// TwinCAT 3 PLC project setpositionGen
// ProgramVersion: 3.1.4020.4
// libraries:
//   Tc2_MC2, * (Beckhoff Automation GmbH)
//   Tc2_Standard, * (Beckhoff Automation GmbH)
//   Tc2_System, * (Beckhoff Automation GmbH)
//   Tc2_TcpIp, * (Beckhoff Automation GmbH)
//   Tc3_Module, * (Beckhoff Automation GmbH)
// project tree:
//   DUTs/ state.TcDUT
//   GVLs/ GVL.TcGVL
//   / PlcTask.TcTTO
//   POUs/ MAIN.TcPOU, TCPServer.TcPOU
// real-time tasks:
//   TASK PlcTask: cycle T#4ms, priority 20, ADS port 350
// motion (NC):
//   TASK NC-Task 1 SAF: cycle T#4ms, priority 4, ADS port 501
//   TASK NC-Task 1 SVB: cycle T#2ms, priority 8, ADS port 511
//   AXIS Axis 1 (id 1)
//     General: UnitName=°
//     Dynamic: AccelerationMaximum=75000, DecelerationMaximum=75000, Acceleration=10000, Deceleration=10000, Jerk=2000000
//     Velo: RefSearch=100, RefSync=100, SlowManual=50, Fast=500, Maximum=744
//     PositionAreaControl: Enable=false, Range=360
//     TargetPosControl: Range=360, Time=0.01
//     encoder EncType=19
//       EncPara: ScaleFactorNumerator=360, ScaleFactorDenominator=421888, Inverse=true, MaxCount=#xffffffff
//     drive DrvType=16
//       DrvPara: MaxCount=#xffffffff, DriveControlDWord=#x00020000
//         Analog: VeloReferenz=100, TorqueSetpointScale=10
//         TimeComp: TaskDelayCycles=1
//     controller CtrType=1
//       CtrPara: PriorControlFactor=1
//         PosDiffControl: Enable=false, Range=360
//         Observer: BandWidth=20
//   AXIS Axis 2 (id 2)
//     General: UnitName=°
//     Dynamic: AccelerationMaximum=75000, DecelerationMaximum=75000, Acceleration=10000, Deceleration=10000, Jerk=2000000
//     Velo: RefSearch=100, RefSync=100, SlowManual=50, Fast=500, Maximum=744
//     PositionAreaControl: Enable=false, Range=360
//     TargetPosControl: Range=360, Time=0.01
//     encoder EncType=19
//       EncPara: ScaleFactorNumerator=360, ScaleFactorDenominator=421888, Inverse=true, MaxCount=#xffffffff
//     drive DrvType=16
//       DrvPara: MaxCount=#xffffffff, DriveControlDWord=#x00020000
//         Analog: VeloReferenz=100, TorqueSetpointScale=10
//         TimeComp: TaskDelayCycles=1
//     controller CtrType=1
//       CtrPara: PriorControlFactor=1
//         PosDiffControl: Enable=false, Range=360
//         Observer: BandWidth=20
//   AXIS Axis 3 (id 3)
//     General: UnitName=°
//     Dynamic: AccelerationMaximum=75000, DecelerationMaximum=75000, Acceleration=10000, Deceleration=10000, Jerk=2000000
//     Velo: RefSearch=100, RefSync=100, SlowManual=50, Fast=500, Maximum=744
//     PositionAreaControl: Enable=false, Range=360
//     TargetPosControl: Range=360, Time=0.01
//     encoder EncType=19
//       EncPara: ScaleFactorNumerator=360, ScaleFactorDenominator=421888, Inverse=true, MaxCount=#xffffffff
//     drive DrvType=16
//       DrvPara: MaxCount=#xffffffff, DriveControlDWord=#x00020000
//         Analog: VeloReferenz=100, TorqueSetpointScale=10
//         TimeComp: TaskDelayCycles=1
//     controller CtrType=1
//       CtrPara: PriorControlFactor=1
//         PosDiffControl: Enable=false, Range=360
//         Observer: BandWidth=20
//   AXIS Axis 4 (id 4)
//     General: UnitName=°
//     Dynamic: AccelerationMaximum=75000, DecelerationMaximum=75000, Acceleration=10000, Deceleration=10000, Jerk=2000000
//     Velo: RefSearch=100, RefSync=100, SlowManual=50, Fast=500, Maximum=744
//     PositionAreaControl: Enable=false, Range=360
//     TargetPosControl: Range=360, Time=0.01
//     encoder EncType=19
//       EncPara: ScaleFactorNumerator=360, ScaleFactorDenominator=421888, Inverse=true, MaxCount=#xffffffff
//     drive DrvType=16
//       DrvPara: MaxCount=#xffffffff, DriveControlDWord=#x00020000
//         Analog: VeloReferenz=100, TorqueSetpointScale=10
//         TimeComp: TaskDelayCycles=1
//     controller CtrType=1
//       CtrPara: PriorControlFactor=1
//         PosDiffControl: Enable=false, Range=360
//         Observer: BandWidth=20
// I/O:
//   DEVICE Device 3 (EtherCAT), AmsNetId 192.168.89.136.4.1
//     Drive 1 (Elmo Drive ) [Gold EtherCAT GCON Drive Rev:0x00010420]
//     Drive 2 (Elmo Drive ) [Gold EtherCAT GCON Drive Rev:0x00010420]
//     Drive 3 (Elmo Drive ) [Gold EtherCAT GCON Drive Rev:0x00010420]
//     Drive 4 (Elmo Drive ) [Gold EtherCAT GCON Drive Rev:0x00010420]
// variable links:
//   NC-Task 1 SAF/Axes/Axis 1 <-> Device 3 (EtherCAT)/Drive 1 (Elmo Drive )
//     Drive/Inputs/In/nDcOutputTime <-> InfoData/DcOutputShift
//     Drive/Inputs/In/nState1 <-> Inputs/Status word
//     Drive/Inputs/In/nState2 <-> Inputs/Status word @bit 8
//     Drive/Inputs/In/nState4 @bit 1 <-> WcState/InputToggle
//     Drive/Inputs/In/nState4 <-> WcState/WcState
//     Drive/Outputs/Out/nCtrl1 <-> Outputs/Control word
//     Drive/Outputs/Out/nCtrl2 <-> Outputs/Control word @bit 8
//     Drive/Outputs/Out/nDataOut1 <-> Outputs/Target Position
//     Enc/Inputs/In/nDataIn1 <-> Inputs/Position actual value
//     Enc/Inputs/In/nDcInputTime <-> InfoData/DcInputShift
//     Enc/Inputs/In/nState4 @bit 1 <-> WcState/InputToggle
//     Enc/Inputs/In/nState4 <-> WcState/WcState
//   NC-Task 1 SAF/Axes/Axis 2 <-> Device 3 (EtherCAT)/Drive 2 (Elmo Drive )
//     Drive/Inputs/In/nDcOutputTime <-> InfoData/DcOutputShift
//     Drive/Inputs/In/nState1 <-> Inputs/Status word
//     Drive/Inputs/In/nState2 <-> Inputs/Status word @bit 8
//     Drive/Inputs/In/nState4 @bit 1 <-> WcState/InputToggle
//     Drive/Inputs/In/nState4 <-> WcState/WcState
//     Drive/Outputs/Out/nCtrl1 <-> Outputs/Control word
//     Drive/Outputs/Out/nCtrl2 <-> Outputs/Control word @bit 8
//     Drive/Outputs/Out/nDataOut1 <-> Outputs/Target Position
//     Enc/Inputs/In/nDataIn1 <-> Inputs/Position actual value
//     Enc/Inputs/In/nDcInputTime <-> InfoData/DcInputShift
//     Enc/Inputs/In/nState4 @bit 1 <-> WcState/InputToggle
//     Enc/Inputs/In/nState4 <-> WcState/WcState
//   NC-Task 1 SAF/Axes/Axis 3 <-> Device 3 (EtherCAT)/Drive 3 (Elmo Drive )
//     Drive/Inputs/In/nDcOutputTime <-> InfoData/DcOutputShift
//     Drive/Inputs/In/nState1 <-> Inputs/Status word
//     Drive/Inputs/In/nState2 <-> Inputs/Status word @bit 8
//     Drive/Inputs/In/nState4 @bit 1 <-> WcState/InputToggle
//     Drive/Inputs/In/nState4 <-> WcState/WcState
//     Drive/Outputs/Out/nCtrl1 <-> Outputs/Control word
//     Drive/Outputs/Out/nCtrl2 <-> Outputs/Control word @bit 8
//     Drive/Outputs/Out/nDataOut1 <-> Outputs/Target Position
//     Enc/Inputs/In/nDataIn1 <-> Inputs/Position actual value
//     Enc/Inputs/In/nDcInputTime <-> InfoData/DcInputShift
//     Enc/Inputs/In/nState4 @bit 1 <-> WcState/InputToggle
//     Enc/Inputs/In/nState4 <-> WcState/WcState
//   NC-Task 1 SAF/Axes/Axis 4 <-> Device 3 (EtherCAT)/Drive 4 (Elmo Drive )
//     Drive/Inputs/In/nDcOutputTime <-> InfoData/DcOutputShift
//     Drive/Inputs/In/nState1 <-> Inputs/Status word
//     Drive/Inputs/In/nState2 <-> Inputs/Status word @bit 8
//     Drive/Inputs/In/nState4 @bit 1 <-> WcState/InputToggle
//     Drive/Inputs/In/nState4 <-> WcState/WcState
//     Drive/Outputs/Out/nCtrl1 <-> Outputs/Control word
//     Drive/Outputs/Out/nCtrl2 <-> Outputs/Control word @bit 8
//     Drive/Outputs/Out/nDataOut1 <-> Outputs/Target Position
//     Enc/Inputs/In/nDataIn1 <-> Inputs/Position actual value
//     Enc/Inputs/In/nDcInputTime <-> InfoData/DcInputShift
//     Enc/Inputs/In/nState4 @bit 1 <-> WcState/InputToggle
//     Enc/Inputs/In/nState4 <-> WcState/WcState
//   setpositionGen/setpositionGen Instance <-> NC-Task 1 SAF/Axes/Axis 1
//     PlcTask Inputs/MAIN.axis1.NcToPlc <-> Outputs/ToPlc
//     PlcTask Outputs/MAIN.axis1.PlcToNc <-> Inputs/FromPlc
//   setpositionGen/setpositionGen Instance <-> NC-Task 1 SAF/Axes/Axis 2
//     PlcTask Inputs/MAIN.axis2.NcToPlc <-> Outputs/ToPlc
//     PlcTask Outputs/MAIN.axis2.PlcToNc <-> Inputs/FromPlc
//   setpositionGen/setpositionGen Instance <-> NC-Task 1 SAF/Axes/Axis 3
//     PlcTask Inputs/MAIN.axis3.NcToPlc <-> Outputs/ToPlc
//     PlcTask Outputs/MAIN.axis3.PlcToNc <-> Inputs/FromPlc
//   setpositionGen/setpositionGen Instance <-> NC-Task 1 SAF/Axes/Axis 4
//     PlcTask Inputs/MAIN.axis4.NcToPlc <-> Outputs/ToPlc
//     PlcTask Outputs/MAIN.axis4.PlcToNc <-> Inputs/FromPlc

CONFIGURATION setpositionGen
    RESOURCE PLC ON TwinCAT3
        TASK PlcTask(INTERVAL := T#4ms, PRIORITY := 20);
        PROGRAM MAIN WITH PlcTask : MAIN;
    END_RESOURCE
END_CONFIGURATION

// ---- DUTs/state.TcDUT

TYPE state :
(
	init := 0,
	gen_power,
	gen_move,
	gen_enable,
	gen_error,
	gen_reset
)INT;
END_TYPE

// ---- GVLs/GVL.TcGVL
{attribute 'qualified_only'}
VAR_GLOBAL
	//数据接收
	Data_receive	   	: ARRAY[1..24]OF BYTE;
	bReceive		   	: BOOL;//接收执行
	rec_busy			:BOOL;
	
	//数据发送
	nSendDataBuffer	   	: ARRAY[1..50]OF BYTE;
	bsend			   	: BOOL;//发送执行
	
	number_recdata      :UDINT;
END_VAR

// ---- POUs/MAIN.TcPOU
PROGRAM MAIN
VAR
	power1,power2,power3,power4: MC_Power;
	axis1,axis2,axis3,axis4: AXIS_REF;
	power1_output,power2_output,power3_output,power4_output:ST_McOutputs;
	

	
	
	move_abs: MC_MoveAbsolute;
	init_pos: LREAL;
	move_init_output:ST_McOutputs;
	
	SetPointGenEnable,SetPointGenEnable1,SetPointGenEnable2,SetPointGenEnable3: MC_ExtSetPointGenEnable;
	SetPointGenDisable,SetPointGenDisable1,SetPointGenDisable2,SetPointGenDisable3: MC_ExtSetPointGenDisable;
	SetPointGenEnable_output,SetPointGenDisable_output,SetPointGenEnable_output1,SetPointGenDisable_output1,SetPointGenEnable_output2,SetPointGenDisable_output2,SetPointGenEnable_output3,SetPointGenDisable_output3:ST_McOutputs;	
	enable,disable:BOOL;
	
	reset_output:ST_McOutputs;
	axis_Reset: MC_Reset;
	
	gen_state:state;
	
	position: LREAL;
	velocity: LREAL;
	direction: DINT;	
	acceleration: LREAL;
	t:LREAL:=0;

	n:UINT:=0;
	a:LINT;
	
	pos1,pos2,pos3,pos4:LREAL;
	acc1,acc2,acc3,acc4:LREAL;
	velo1,velo2,velo3,velo4:LREAL;
	dir: DINT:=1;
	inpos:BOOL:=1;
	flag:UINT:=0;

	flag1: INT;
	ADS_Array: ARRAY[0..12] OF UINT;
	ADS_ParaArray: ARRAY[0..11] OF UINT;
	avar:LREAL;
END_VAR

axis1();(*更新轴状态*)
axis2();(*更新轴状态*)
axis3();(*更新轴状态*)
axis4();(*更新轴状态*)
axis1.ReadStatus();
axis2.ReadStatus();
axis3.ReadStatus();
axis4.ReadStatus();
power();
setpositionGen();
reset();

//move_init();
//TCP/IP receive data
IF NOT GVL.rec_busy THEN
	GVL.bReceive:=TRUE;
END_IF
TCPServer();
IF GVL.number_recdata<>0 THEN
	gen_state:=gen_enable;
	GVL.number_recdata:=0;
	IF GVL.Data_receive[1]>16#7F THEN 
	   GVL.Data_receive[1]:=GVL.Data_receive[1] AND 16#7F;
 	   flag:=1;	
	END_IF
	pos1:=GVL.Data_receive[1];
	pos1:=pos1*256;
	pos1:=(pos1+GVL.Data_receive[2])/10;
	IF flag=1 THEN
		pos1:=-pos1;
		flag:=0;
	END_IF
	velo1:=GVL.Data_receive[3];
	velo1:=velo1*256;
	velo1:=(velo1+GVL.Data_receive[4])/10;
	acc1:=GVL.Data_receive[5];
	acc1:=acc1*256;
	acc1:=(acc1+GVL.Data_receive[6])/10;
	
	IF GVL.Data_receive[7]>16#7F THEN 
	   GVL.Data_receive[7]:=GVL.Data_receive[7] AND 16#7F;
 	   flag:=1;	
	END_IF
	pos2:=GVL.Data_receive[7];
	pos2:=pos2*256;
	pos2:=(pos2+GVL.Data_receive[8])/10;
	IF flag=1 THEN
		pos2:=-pos2;
		flag:=0;
	END_IF
	velo2:=GVL.Data_receive[9];
	velo2:=velo2*256;
	velo2:=(velo2+GVL.Data_receive[10])/10;
	acc2:=GVL.Data_receive[11];
	acc2:=acc2*256;
	acc2:=(acc2+GVL.Data_receive[12])/10;
	
	IF GVL.Data_receive[13]>16#7F THEN 
	   GVL.Data_receive[13]:=GVL.Data_receive[13] AND 16#7F;
 	   flag:=1;	
	END_IF
	pos3:=GVL.Data_receive[13];
	pos3:=pos3*256;
	pos3:=(pos3+GVL.Data_receive[14])/10;
	IF flag=1 THEN
		pos3:=-pos3;
		flag:=0;
	END_IF
	velo3:=GVL.Data_receive[15];
	velo3:=velo3*256;
	velo3:=(velo3+GVL.Data_receive[16])/10;
	acc3:=GVL.Data_receive[17];
	acc3:=acc3*256;
	acc3:=(acc3+GVL.Data_receive[18])/10;
	
	IF GVL.Data_receive[19]>16#7F THEN 
	   GVL.Data_receive[19]:=GVL.Data_receive[19] AND 16#7F;
 	   flag:=1;	
	END_IF
	pos4:=GVL.Data_receive[19];
	pos4:=pos4*256;
	pos4:=(pos4+GVL.Data_receive[20])/10;
	IF flag=1 THEN
		pos4:=-pos4;
		flag:=0;
	END_IF
	velo4:=GVL.Data_receive[21];
	velo4:=velo4*256;
	velo4:=(velo4+GVL.Data_receive[22])/10;
	acc4:=GVL.Data_receive[23];
	acc4:=acc4*256;
	acc4:=(acc4+GVL.Data_receive[24])/10;
END_IF

//ADS receive data
IF ADS_Array[12]=1 THEN
	ADS_Array[12]:=0;
	gen_state:=gen_enable;
	pos1:=ADS_Array[0];
	pos1:=pos1/10;
	velo1:=ADS_Array[1];
	velo1:=velo1/10;
	acc1:=ADS_Array[2];
	acc1:=acc1/10;
	pos2:=ADS_Array[3];
	pos2:=pos2/10;
	velo2:=ADS_Array[4];
	velo2:=velo2/10;
	acc2:=ADS_Array[5];
	acc2:=acc2/10;
	pos3:=ADS_Array[6];
	pos3:=pos3/10;
	velo3:=ADS_Array[7];
	velo3:=velo3/10;
	acc3:=ADS_Array[8];
	acc3:=acc3/10;
	pos4:=ADS_Array[9];
	pos4:=pos4/10;
	velo4:=ADS_Array[10];
	velo4:=velo4/10;
	acc4:=ADS_Array[11];
	acc4:=acc4/10;
END_IF
//ADS updata
avar:=axis1.NcToPlc.ActPos;  //位置
avar:=avar*10;
ADS_ParaArray[0]:= TO_UINT(avar);
avar:=axis1.NcToPlc.Actvelo;  //速度
avar:=avar*10;
ADS_ParaArray[1]:=TO_UINT(avar);
avar:=axis1.NcToPlc.ActAcc;  //加速度
avar:=avar*10;
ADS_ParaArray[2]:=TO_UINT(avar);

avar:=axis2.NcToPlc.ActPos;  //位置
avar:=avar*10;
ADS_ParaArray[3]:= TO_UINT(avar);
avar:=axis2.NcToPlc.Actvelo;  //速度
avar:=avar*10;
ADS_ParaArray[4]:=TO_UINT(avar);
avar:=axis2.NcToPlc.ActAcc;  //加速度
avar:=avar*10;
ADS_ParaArray[5]:=TO_UINT(avar);

avar:=axis3.NcToPlc.ActPos;  //位置
avar:=avar*10;
ADS_ParaArray[6]:= TO_UINT(avar);
avar:=axis3.NcToPlc.Actvelo;  //速度
avar:=avar*10;
ADS_ParaArray[7]:=TO_UINT(avar);
avar:=axis3.NcToPlc.ActAcc;  //加速度
avar:=avar*10;
ADS_ParaArray[8]:=TO_UINT(avar);

avar:=axis4.NcToPlc.ActPos;  //位置
avar:=avar*10;
ADS_ParaArray[9]:= TO_UINT(avar);
avar:=axis4.NcToPlc.Actvelo;  //速度
avar:=avar*10;
ADS_ParaArray[10]:=TO_UINT(avar);
avar:=axis4.NcToPlc.ActAcc;  //加速度
avar:=avar*10;
ADS_ParaArray[11]:=TO_UINT(avar);

CASE gen_state OF
	init:
		power1.Enable:=FALSE;
		power2.Enable:=FALSE;
		power3.Enable:=FALSE;
		power4.Enable:=FALSE;
		SetPointGenEnable.Execute:=FALSE;
		SetPointGenDisable.Execute:=FALSE;
		SetPointGenEnable1.Execute:=FALSE;
		SetPointGenDisable1.Execute:=FALSE;
		SetPointGenEnable2.Execute:=FALSE;
		SetPointGenDisable2.Execute:=FALSE;
		SetPointGenEnable3.Execute:=FALSE;
		SetPointGenDisable3.Execute:=FALSE;
		axis_Reset.Execute:=FALSE;
		gen_state:=gen_power;
			
	gen_power:
		power1.Enable:=TRUE;
		power2.Enable:=TRUE;
		power3.Enable:=TRUE;
		power4.Enable:=TRUE;
		IF power1_output.Done AND power2_output.Done AND power3_output.Done AND power4_output.Done THEN
			gen_state:=gen_move;
		END_IF
		IF axis1.Status.Error OR axis2.Status.Error OR axis3.Status.Error OR axis4.Status.Error THEN
			gen_state := gen_error;
		END_IF
		
	gen_move:
		//	gen_state:=gen_enable;
	gen_enable:

		setpointgenenable.Execute:=TRUE;
		setpointgenenable1.Execute:=TRUE;
		setpointgenenable2.Execute:=TRUE;
		setpointgenenable3.Execute:=TRUE;
		IF SetPointGenEnable.Enabled AND SetPointGenEnable1.Enabled AND SetPointGenEnable2.Enabled AND SetPointGenEnable3.Enabled AND inpos THEN
			flag:=1;
		END_IF

		IF flag=1 THEN
			gen_state:=gen_move;
			IF velo1>1 THEN
				MC_ExtSetPointGenFeed(
					Position:= pos1,		
					Velocity:= velo1, 
					Acceleration:=acc1, 
					Direction:= dir,
					Axis:= axis1);	
			END_IF
			IF velo2>1 THEN
				MC_ExtSetPointGenFeed(
					Position:= pos2,		
					Velocity:= velo2, 
					Acceleration:=acc2, 
					Direction:= dir,
					Axis:= axis2);	
			END_IF
			IF velo3>1 THEN
				MC_ExtSetPointGenFeed(
					Position:= pos3,		
					Velocity:= velo3, 
					Acceleration:=acc3, 
					Direction:= dir,
					Axis:= axis3);
			END_IF	
			IF velo4>1 THEN
				MC_ExtSetPointGenFeed(
					Position:= pos4,		
					Velocity:= velo4, 
					Acceleration:=acc4, 
					Direction:= dir,
					Axis:= axis4);
			END_IF	
		END_IF
		
	//	IF axis1.Status.InTargetPosition AND axis2.Status.InTargetPosition AND axis3.Status.InTargetPosition AND axis4.Status.InTargetPosition AND flag=0 THEN
	//		inpos:=TRUE;
	//	END_IF
		
		IF flag=1 THEN
			flag:=0;
		END_IF

		IF axis1.Status.Error THEN
			gen_state := gen_error;
		END_IF
	
	gen_error:
		SetPointGenEnable.Execute:=FALSE;
		SetPointGenDisable.Execute := SetPointGenEnable.Enabled;	
		SetPointGenEnable1.Execute:=FALSE;
		SetPointGenDisable1.Execute := SetPointGenEnable1.Enabled;
		IF NOT axis1.Status.Coupled THEN
			IF axis1.Status.Error THEN
				gen_state := gen_reset;	
			ELSE
				gen_state := init;
			END_IF
		END_IF
	
	gen_reset:
		axis_Reset.Execute := TRUE;
		SetPointGenDisable.Execute:=FALSE;
		SetPointGenDisable1.Execute:=FALSE;
			
			IF axis_Reset.Done  THEN
				gen_state := init;
			ELSIF axis_Reset.Error  THEN
				gen_state := init; 
			END_IF
		
END_CASE

ACTION move_init:
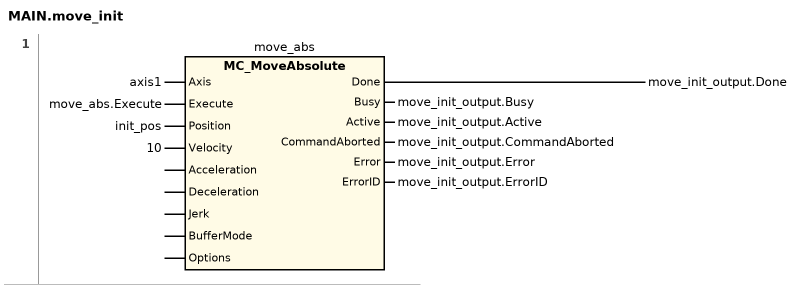
// NETWORK 1
move_abs(
    Axis := axis1,
    Execute := move_abs.Execute,
    Position := init_pos,
    Velocity := 10,
    Busy => move_init_output.Busy,
    Active => move_init_output.Active,
    CommandAborted => move_init_output.CommandAborted,
    Error => move_init_output.Error,
    ErrorID => move_init_output.ErrorID); // MC_MoveAbsolute
move_init_output.Done := move_abs.Done;
END_ACTION

ACTION power:
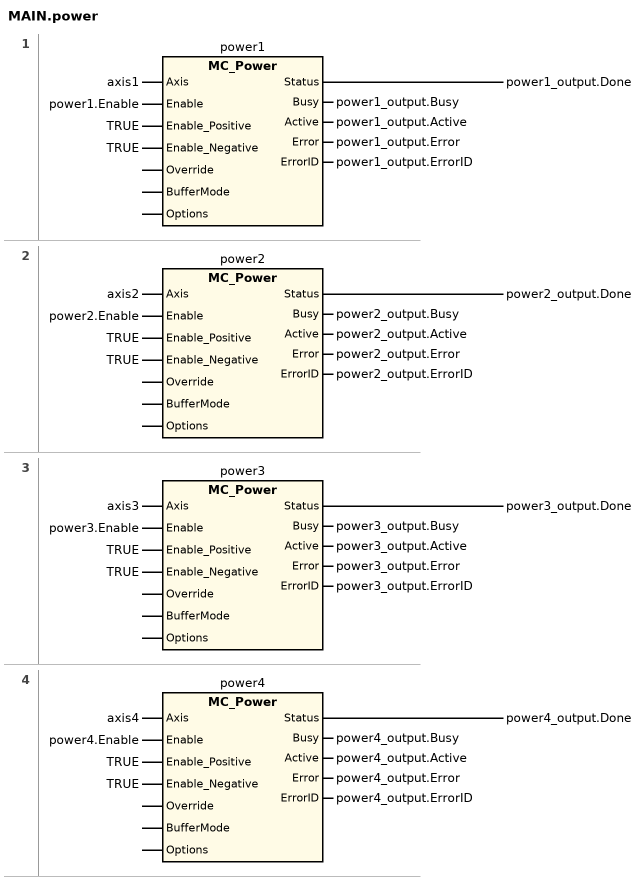
// NETWORK 1
power1(
    Axis := axis1,
    Enable := power1.Enable,
    Enable_Positive := TRUE,
    Enable_Negative := TRUE,
    Busy => power1_output.Busy,
    Active => power1_output.Active,
    Error => power1_output.Error,
    ErrorID => power1_output.ErrorID); // MC_Power
power1_output.Done := power1.Status;

// NETWORK 2
power2(
    Axis := axis2,
    Enable := power2.Enable,
    Enable_Positive := TRUE,
    Enable_Negative := TRUE,
    Busy => power2_output.Busy,
    Active => power2_output.Active,
    Error => power2_output.Error,
    ErrorID => power2_output.ErrorID); // MC_Power
power2_output.Done := power2.Status;

// NETWORK 3
power3(
    Axis := axis3,
    Enable := power3.Enable,
    Enable_Positive := TRUE,
    Enable_Negative := TRUE,
    Busy => power3_output.Busy,
    Active => power3_output.Active,
    Error => power3_output.Error,
    ErrorID => power3_output.ErrorID); // MC_Power
power3_output.Done := power3.Status;

// NETWORK 4
power4(
    Axis := axis4,
    Enable := power4.Enable,
    Enable_Positive := TRUE,
    Enable_Negative := TRUE,
    Busy => power4_output.Busy,
    Active => power4_output.Active,
    Error => power4_output.Error,
    ErrorID => power4_output.ErrorID); // MC_Power
power4_output.Done := power4.Status;
END_ACTION

ACTION reset:
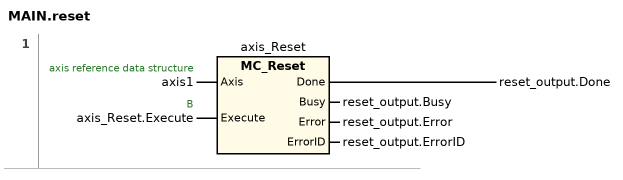
// NETWORK 1
//   axis1: axis reference data structure
//   axis_Reset.Execute: B
axis_Reset(
    Axis := axis1,
    Execute := axis_Reset.Execute,
    Busy => reset_output.Busy,
    Error => reset_output.Error,
    ErrorID => reset_output.ErrorID); // MC_Reset
reset_output.Done := axis_Reset.Done;
END_ACTION

ACTION setpositionGen:
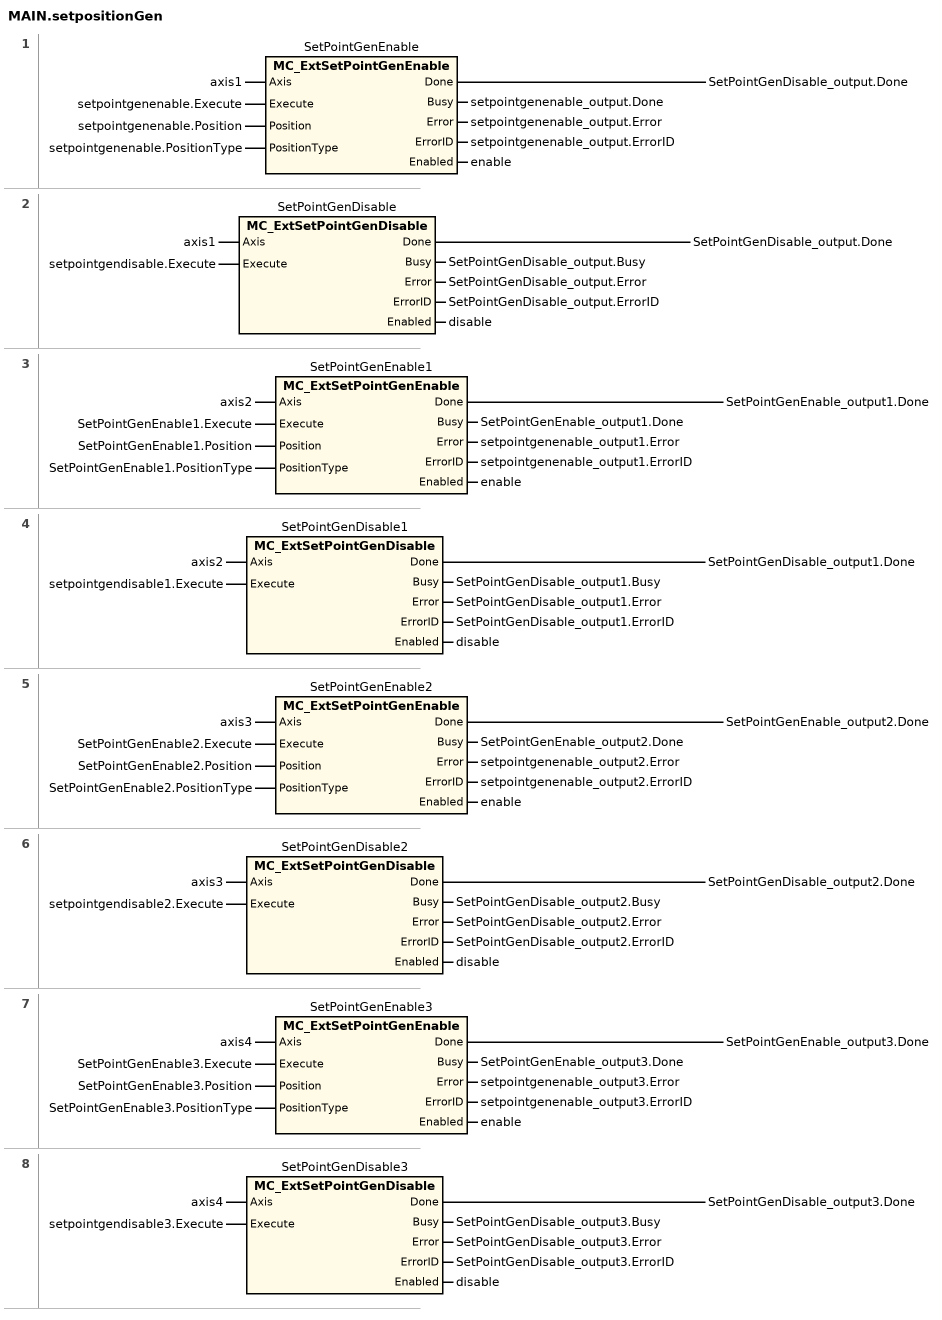
// NETWORK 1
SetPointGenEnable(
    Axis := axis1,
    Execute := setpointgenenable.Execute,
    Position := setpointgenenable.Position,
    PositionType := setpointgenenable.PositionType,
    Busy => setpointgenenable_output.Done,
    Error => setpointgenenable_output.Error,
    ErrorID => setpointgenenable_output.ErrorID,
    Enabled => enable); // MC_ExtSetPointGenEnable
SetPointGenDisable_output.Done := SetPointGenEnable.Done;

// NETWORK 2
SetPointGenDisable(
    Axis := axis1,
    Execute := setpointgendisable.Execute,
    Busy => SetPointGenDisable_output.Busy,
    Error => SetPointGenDisable_output.Error,
    ErrorID => SetPointGenDisable_output.ErrorID,
    Enabled => disable); // MC_ExtSetPointGenDisable
SetPointGenDisable_output.Done := SetPointGenDisable.Done;

// NETWORK 3
SetPointGenEnable1(
    Axis := axis2,
    Execute := SetPointGenEnable1.Execute,
    Position := SetPointGenEnable1.Position,
    PositionType := SetPointGenEnable1.PositionType,
    Busy => SetPointGenEnable_output1.Done,
    Error => setpointgenenable_output1.Error,
    ErrorID => setpointgenenable_output1.ErrorID,
    Enabled => enable); // MC_ExtSetPointGenEnable
SetPointGenEnable_output1.Done := SetPointGenEnable1.Done;

// NETWORK 4
SetPointGenDisable1(
    Axis := axis2,
    Execute := setpointgendisable1.Execute,
    Busy => SetPointGenDisable_output1.Busy,
    Error => SetPointGenDisable_output1.Error,
    ErrorID => SetPointGenDisable_output1.ErrorID,
    Enabled => disable); // MC_ExtSetPointGenDisable
SetPointGenDisable_output1.Done := SetPointGenDisable1.Done;

// NETWORK 5
SetPointGenEnable2(
    Axis := axis3,
    Execute := SetPointGenEnable2.Execute,
    Position := SetPointGenEnable2.Position,
    PositionType := SetPointGenEnable2.PositionType,
    Busy => SetPointGenEnable_output2.Done,
    Error => setpointgenenable_output2.Error,
    ErrorID => setpointgenenable_output2.ErrorID,
    Enabled => enable); // MC_ExtSetPointGenEnable
SetPointGenEnable_output2.Done := SetPointGenEnable2.Done;

// NETWORK 6
SetPointGenDisable2(
    Axis := axis3,
    Execute := setpointgendisable2.Execute,
    Busy => SetPointGenDisable_output2.Busy,
    Error => SetPointGenDisable_output2.Error,
    ErrorID => SetPointGenDisable_output2.ErrorID,
    Enabled => disable); // MC_ExtSetPointGenDisable
SetPointGenDisable_output2.Done := SetPointGenDisable2.Done;

// NETWORK 7
SetPointGenEnable3(
    Axis := axis4,
    Execute := SetPointGenEnable3.Execute,
    Position := SetPointGenEnable3.Position,
    PositionType := SetPointGenEnable3.PositionType,
    Busy => SetPointGenEnable_output3.Done,
    Error => setpointgenenable_output3.Error,
    ErrorID => setpointgenenable_output3.ErrorID,
    Enabled => enable); // MC_ExtSetPointGenEnable
SetPointGenEnable_output3.Done := SetPointGenEnable3.Done;

// NETWORK 8
SetPointGenDisable3(
    Axis := axis4,
    Execute := setpointgendisable3.Execute,
    Busy => SetPointGenDisable_output3.Busy,
    Error => SetPointGenDisable_output3.Error,
    ErrorID => SetPointGenDisable_output3.ErrorID,
    Enabled => disable); // MC_ExtSetPointGenDisable
SetPointGenDisable_output3.Done := SetPointGenDisable3.Done;
END_ACTION

END_PROGRAM

// ---- POUs/TCPServer.TcPOU
PROGRAM TCPServer
VAR	
	bSuccess					: BOOL;//函数 F_CreateServerHnd 用于初始化句柄 hServer 内部参数并创建服务器，bSuccess确认是否建立成功
	bEnable						: BOOL;//是否启用
	Step						: INT;
	iCount						: INT;

	//控制器做 TCPIP 的 Server
	sRemoteHost 				: STRING(15) := '169.254.130.170';//控制器IP地址
	nRemotePort 				: UDINT := 2000;//控制器端口号
	fb_ServerConnection			: FB_ServerClientConnection;//建立server 和client连接
	hServer						: T_HSERVER;//TCPIP被创建的服务器
	hSocket						: T_HSOCKET;//TCPIP句柄

	//数据接收
	fb_Receive					: FB_SocketReceive;
//	Data_receive	   AT%Q*	: ARRAY[1..10]OF BYTE;
//	bReceive		   AT%I*	: BOOL;//接收执行
	
	//数据发送
	fb_Send						: FB_SocketSend;
//	nSendDataBuffer	   AT%I*	: ARRAY[1..50]OF BYTE;
//	bsend			   AT%I*	: BOOL;//发送执行
END_VAR

FBD();
CASE step OF
0:
	bSuccess:=FALSE;
    bEnable:=FALSE;
         step:=step+1;
1:
	bSuccess:=F_CreateServerHnd(
	sSrvNetID:='' ,
	sLocalHost:=sRemoteHost ,
	nLocalPort:=nRemotePort ,
	nMode:=LISTEN_MODE_CLOSEALL OR CONNECT_MODE_ENABLEDBG ,
	bEnable:=TRUE ,
	hServer:=hserver );
         step:=step+1;

2:
        IF bSuccess THEN
 	       bEnable:=TRUE;
	        IF  NOT fb_ServerConnection.bError THEN
		          step:=step+1;
	         ELSE
 		        step:=0;
   	      	END_IF
      	ELSE
	         step:=0;
      	END_IF

3:
		IF fb_ServerConnection.eState=eSOCKET_CONNECTED THEN
				iCount:=iCount+1;
 				step:=step+1;
		END_IF

4:

    fb_Receive(
	sSrvNetId:='' ,
	hSocket:=hSocket ,
	cbLen:=SIZEOF(GVL.Data_receive) ,
	pDest:=ADR(GVL.Data_receive) ,
	bExecute:=GVL.bReceive ,
	tTimeout:=T#1S ,
	bBusy=> ,
	bError=> ,
	nErrId=> ,
	nRecBytes=> );
IF   NOT fb_Receive.bbusy OR NOT fb_Receive.berror THEN
	fb_Send(
	sSrvNetId:='' ,
	hSocket:=hSocket ,
	cbLen:=SIZEOF(GVL.nSendDataBuffer) ,
	pSrc:=ADR(GVL.nSendDataBuffer) ,
	bExecute:=GVL.bsend ,
	tTimeout:=t#6s ,
	bBusy=> ,
	bError=> ,
	nErrId=> );
END_IF
//		ELSE
//   		 step:=0;
GVL.rec_busy:=fb_Receive.bBusy;
IF fb_Receive.nRecBytes>0 THEN
			GVL.number_recdata:=fb_Receive.nRecBytes;//返回接收到的数据个数
END_IF	
IF GVL.bReceive=TRUE THEN
			GVL.bReceive:=FALSE;//只接收一次数据
END_IF
IF GVL.bsend=TRUE THEN
			GVL.bsend:=FALSE;//只发送一次数据
END_IF
END_CASE

ACTION FBD:
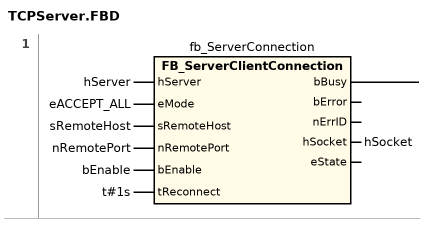
// NETWORK 1
fb_ServerConnection(
    hServer := hServer,
    eMode := eACCEPT_ALL,
    sRemoteHost := sRemoteHost,
    nRemotePort := nRemotePort,
    bEnable := bEnable,
    tReconnect := t#1s,
    hSocket => hSocket); // FB_ServerClientConnection
END_ACTION

END_PROGRAM
